Staubli VAL3: iLevel2.pgx

public program iLevel2(num& nNum[] (dimensions=1))
begin
  nNum=dioGet(iLevel2)
end
